(* OutputValue := InputValue * (OutputMax - OutputMin)/(InputMax - InputMin) + OutputMin *)
FUNCTION_BLOCK AnalogScaleWithAlarm
VAR_INPUT
	InputValue	: LREAL;
	InputMin	: LREAL:=0;
	InputMax	: LREAL:=100;
	OutputMin	: LREAL:=0;
	OutputMax	: LREAL:=100;
	LL_Set	: LREAL;
	L_Set	: LREAL;
	H_Set	: LREAL;
	HH_Set	: LREAL;
END_VAR
VAR_OUTPUT
	OutputValue	: LREAL;
	Percentage : LREAL;
	DataInvalid : BOOL;
	LL : BOOL;
	L : BOOL;
	H : BOOL;
	HH : BOOL;
END_VAR
VAR
END_VAR

IF InputMax - InputMin = 0 THEN
	DataInvalid := TRUE;
ELSE
	OutputValue := InputValue * (OutputMax - OutputMin)/(InputMax - InputMin) + OutputMin;
	Percentage := (InputValue - InputMin)/(InputMax - InputMin);
	DataInvalid := FALSE;
END_IF

LL := OutputValue < LL_Set;
L := OutputValue < L_Set;
H := OutputValue > H_Set;
HH := OutputValue > HH_Set;

END_FUNCTION_BLOCK

(* stored: Version 1.1.0.1, ProductVersion 3.1.4024.12
   POU AnalogScaleWithAlarm: Id {af70b0ba-e473-435d-b244-219eb065e0de}, SpecialFunc None *)
